FUNCTION_BLOCK FB_Hmi_Switch
VAR_INPUT
END_VAR
VAR_OUTPUT
END_VAR
VAR
END_VAR

END_FUNCTION_BLOCK

(* stored: Version 1.1.0.1, ProductVersion 3.1.4024.10
   POU FB_Hmi_Switch: Id {062b3d7f-a5f8-426d-b207-093b1ba420c0}, SpecialFunc None *)
